# EPICS substitutions: epm2000App/Db/epm2000.substitutions
file epm2000chan.template
{
pattern { dev     ,ch     , QM   , thr_enable ,     DESC    }
        { $(cha)  , A     , "\'" ,    $(chath),  $(desc_a)  }
        { $(chb)  , B     , "\'" ,    $(chbth),  $(desc_b)  }
}

file epm2000cont.template
{
pattern { dev         , QM    }
        { $(cont)     , "\'"  }
}
